ADAPTER IAIStatus (* Adapter Interface *)
  (* Standard: 61499-1 *)
  (* Version 0.0, 3/4/2026, Schneider Electric *)
  PACKAGE SE.Nereda;
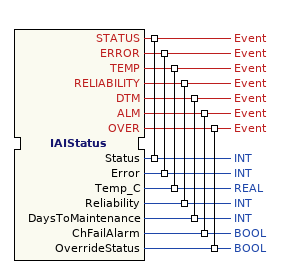
  EVENT_OUTPUT
    STATUS WITH Status; (* Confirmation from Plug *)
    ERROR WITH Error;
    TEMP WITH Temp_C;
    RELIABILITY WITH Reliability;
    DTM WITH DaysToMaintenance;
    ALM WITH ChFailAlarm;
    OVER WITH OverrideStatus;
  END_EVENT
  VAR_OUTPUT
    Status : INT;
    Error : INT;
    Temp_C : REAL;
    Reliability : INT;
    DaysToMaintenance : INT;
    ChFailAlarm : BOOL;
    OverrideStatus : BOOL;
  END_VAR
  SERVICE SOCKET/PLUG
    SEQUENCE request_confirm
      SOCKET.REQ(REQD) -> PLUG.REQ(REQD);
      PLUG.STATUS(CNFD) -> SOCKET.STATUS(CNFD);
    END_SEQUENCE
    SEQUENCE indication_response
      PLUG.IND(INDD) -> SOCKET.IND(INDD);
      SOCKET.RSP(RSPD) -> PLUG.RSP(RSPD);
    END_SEQUENCE
  END_SERVICE
END_ADAPTER
